# EPICS substitutions: siteApps/alarmPerfTest/alarmTestApp/Db/alarm.substitutions
###############################
file "$(DB_TOP)/alarm.template" { pattern
{S,				VAL}
{Alarm0,			92.30}
{Alarm1,			95.71}
{Alarm2,			98.12}
{Alarm3,			91.53}
{Alarm4,			94.94}
{Alarm5,			97.35}
{Alarm6,			90.76}
{Alarm7,			93.17}
{Alarm8,			96.58}
{Alarm9,			99.99}
{Alarm10,			92.30}
{Alarm11,			95.71}
{Alarm12,			98.12}
{Alarm13,			91.53}
{Alarm14,			94.94}
{Alarm15,			97.35}
{Alarm16,			90.76}
{Alarm17,			93.17}
{Alarm18,			96.58}
{Alarm19,			99.99}
{Alarm20,			92.30}
{Alarm21,			95.71}
{Alarm22,			98.12}
{Alarm23,			91.53}
{Alarm24,			94.94}
{Alarm25,			97.35}
{Alarm26,			90.76}
{Alarm27,			93.17}
{Alarm28,			96.58}
{Alarm29,			99.99}
{Alarm30,			92.30}
{Alarm31,			95.71}
{Alarm32,			98.02}
{Alarm33,			91.03}
{Alarm34,			94.04}
{Alarm35,			97.15}
{Alarm36,			90.16}
{Alarm37,			93.27}
{Alarm38,			96.28}
{Alarm39,			99.29}
{Alarm40,			92.20}
{Alarm41,			95.21}
{Alarm42,			98.32}
{Alarm43,			91.33}
{Alarm44,			99.34}
{Alarm45,			99.45}
{Alarm46,			90.46}
{Alarm47,			93.57}
{Alarm48,			96.58}
{Alarm49,			99.59}
{Alarm50,			92.50}
{Alarm51,			95.51}
{Alarm52,			98.62}
{Alarm53,			91.63}
{Alarm54,			94.64}
{Alarm55,			97.75}
{Alarm56,			90.76}
{Alarm57,			93.87}
{Alarm58,			96.88}
{Alarm59,			99.89}
{Alarm60,			92.80}
{Alarm61,			95.81}
{Alarm62,			98.92}
{Alarm63,			91.93}
{Alarm64,			94.94}
{Alarm65,			97.05}
{Alarm66,			90.06}
{Alarm67,			93.17}
{Alarm68,			96.18}
{Alarm69,			99.19}
{Alarm70,			92.10}
{Alarm71,			95.11}
{Alarm72,			98.22}
{Alarm73,			91.23}
{Alarm74,			94.24}
{Alarm75,			97.35}
{Alarm76,			90.36}
{Alarm77,			93.47}
{Alarm78,			96.48}
{Alarm79,			99.49}
{Alarm80,			92.40}
{Alarm81,			95.41}
{Alarm82,			98.52}
{Alarm83,			91.53}
{Alarm84,			94.54}
{Alarm85,			97.65}
{Alarm86,			90.66}
{Alarm87,			93.77}
{Alarm88,			96.78}
{Alarm89,			99.79}
{Alarm90,			92.70}
{Alarm91,			95.71}
{Alarm92,			98.82}
{Alarm93,			91.83}
{Alarm94,			94.84}
{Alarm95,			97.95}
{Alarm96,			90.96}
{Alarm97,			93.07}
{Alarm98,			96.08}
{Alarm99,			99.09}
{Alarm100,			92.00}
{Alarm101,			95.01}
{Alarm102,			98.12}
{Alarm103,			91.13}
{Alarm104,			94.14}
{Alarm105,			97.25}
{Alarm106,			90.26}
{Alarm107,			93.37}
{Alarm108,			96.38}
{Alarm109,			99.39}
{Alarm110,			92.30}
{Alarm111,			95.31}
{Alarm112,			98.42}
{Alarm113,			91.43}
{Alarm114,			94.44}
{Alarm115,			97.55}
{Alarm116,			90.56}
{Alarm117,			93.67}
{Alarm118,			96.68}
{Alarm119,			99.69}
{Alarm120,			92.60}
{Alarm121,			95.61}
{Alarm122,			98.72}
{Alarm123,			91.73}
{Alarm124,			94.74}
{Alarm125,			97.85}
{Alarm126,			90.86}
{Alarm127,			93.97}
{Alarm128,			96.98}
{Alarm129,			99.99}
{Alarm130,			92.90}
{Alarm131,			95.91}
{Alarm132,			98.02}
{Alarm133,			91.03}
{Alarm134,			94.04}
{Alarm135,			97.15}
{Alarm136,			90.16}
{Alarm137,			93.27}
{Alarm138,			96.28}
{Alarm139,			99.29}
{Alarm140,			92.20}
{Alarm141,			95.21}
{Alarm142,			98.32}
{Alarm143,			91.33}
{Alarm144,			94.34}
{Alarm145,			97.45}
{Alarm146,			90.46}
{Alarm147,			93.57}
{Alarm148,			96.58}
{Alarm149,			99.59}
{Alarm150,			92.50}
{Alarm151,			95.51}
{Alarm152,			98.62}
{Alarm153,			91.63}
{Alarm154,			94.64}
{Alarm155,			97.75}
{Alarm156,			90.76}
{Alarm157,			93.87}
{Alarm158,			96.88}
{Alarm159,			99.89}
{Alarm160,			92.80}
{Alarm161,			95.81}
{Alarm162,			98.92}
{Alarm163,			91.93}
{Alarm164,			94.94}
{Alarm165,			97.05}
{Alarm166,			90.06}
{Alarm167,			93.17}
{Alarm168,			96.18}
{Alarm169,			99.19}
{Alarm170,			92.10}
{Alarm171,			95.11}
{Alarm172,			98.22}
{Alarm173,			91.23}
{Alarm174,			94.24}
{Alarm175,			97.35}
{Alarm176,			90.36}
{Alarm177,			93.47}
{Alarm178,			96.48}
{Alarm179,			99.49}
{Alarm180,			92.40}
{Alarm181,			95.41}
{Alarm182,			98.52}
{Alarm183,			91.53}
{Alarm184,			94.54}
{Alarm185,			97.65}
{Alarm186,			90.66}
{Alarm187,			93.77}
{Alarm188,			96.78}
{Alarm189,			99.79}
{Alarm190,			92.70}
{Alarm191,			95.71}
{Alarm192,			98.82}
{Alarm193,			91.83}
{Alarm194,			94.84}
{Alarm195,			97.95}
{Alarm196,			90.96}
{Alarm197,			93.07}
{Alarm198,			96.08}
{Alarm199,			99.09}
{Alarm200,			92.00}
{Alarm201,			95.01}
{Alarm202,			98.12}
{Alarm203,			91.13}
{Alarm204,			94.14}
{Alarm205,			97.25}
{Alarm206,			90.26}
{Alarm207,			93.37}
{Alarm208,			96.38}
{Alarm209,			99.39}
{Alarm210,			92.30}
{Alarm211,			95.31}
{Alarm212,			98.42}
{Alarm213,			91.43}
{Alarm214,			94.44}
{Alarm215,			97.55}
{Alarm216,			90.56}
{Alarm217,			93.67}
{Alarm218,			96.68}
{Alarm219,			99.69}
{Alarm220,			92.60}
{Alarm221,			95.61}
{Alarm222,			98.72}
{Alarm223,			91.73}
{Alarm224,			94.74}
{Alarm225,			97.85}
{Alarm226,			90.86}
{Alarm227,			93.97}
{Alarm228,			96.98}
{Alarm229,			99.99}
{Alarm230,			92.90}
{Alarm231,			95.91}
{Alarm232,			98.02}
{Alarm233,			91.03}
{Alarm234,			94.04}
{Alarm235,			97.15}
{Alarm236,			90.16}
{Alarm237,			93.27}
{Alarm238,			96.28}
{Alarm239,			99.29}
{Alarm240,			92.20}
{Alarm241,			95.21}
{Alarm242,			98.32}
{Alarm243,			91.33}
{Alarm244,			94.34}
{Alarm245,			97.45}
{Alarm246,			90.46}
{Alarm247,			93.57}
{Alarm248,			96.58}
{Alarm249,			99.59}
{Alarm250,			92.50}
{Alarm251,			95.51}
{Alarm252,			98.62}
{Alarm253,			91.63}
{Alarm254,			94.64}
{Alarm255,			97.75}
{Alarm256,			90.76}
{Alarm257,			93.87}
{Alarm258,			96.88}
{Alarm259,			99.89}
{Alarm260,			92.80}
{Alarm261,			95.81}
{Alarm262,			98.92}
{Alarm263,			91.93}
{Alarm264,			94.94}
{Alarm265,			97.05}
{Alarm266,			90.06}
{Alarm267,			93.17}
{Alarm268,			96.18}
{Alarm269,			99.19}
{Alarm270,			92.10}
{Alarm271,			95.11}
{Alarm272,			98.22}
{Alarm273,			91.23}
{Alarm274,			94.24}
{Alarm275,			97.35}
{Alarm276,			90.36}
{Alarm277,			93.47}
{Alarm278,			96.48}
{Alarm279,			99.49}
{Alarm280,			92.40}
{Alarm281,			95.41}
{Alarm282,			98.52}
{Alarm283,			91.53}
{Alarm284,			94.54}
{Alarm285,			97.65}
{Alarm286,			90.66}
{Alarm287,			93.77}
{Alarm288,			96.78}
{Alarm289,			99.79}
{Alarm290,			92.70}
{Alarm291,			95.71}
{Alarm292,			98.82}
{Alarm293,			91.83}
{Alarm294,			94.84}
{Alarm295,			97.95}
{Alarm296,			90.96}
{Alarm297,			93.07}
{Alarm298,			96.08}
{Alarm299,			99.09}
{Alarm300,			92.00}
{Alarm301,			95.01}
{Alarm302,			98.12}
{Alarm303,			91.13}
{Alarm304,			94.14}
{Alarm305,			97.25}
{Alarm306,			90.26}
{Alarm307,			93.37}
{Alarm308,			96.38}
{Alarm309,			99.39}
{Alarm310,			92.30}
{Alarm311,			95.31}
{Alarm312,			98.42}
{Alarm313,			91.43}
{Alarm314,			94.44}
{Alarm315,			97.55}
{Alarm316,			90.56}
{Alarm317,			93.67}
{Alarm318,			96.68}
{Alarm319,			99.69}
{Alarm320,			92.60}
{Alarm321,			95.61}
{Alarm322,			98.72}
{Alarm323,			91.73}
{Alarm324,			94.74}
{Alarm325,			97.85}
{Alarm326,			90.86}
{Alarm327,			93.97}
{Alarm328,			96.98}
{Alarm329,			99.99}
{Alarm330,			92.90}
{Alarm331,			95.91}
{Alarm332,			98.12}
{Alarm333,			91.53}
{Alarm334,			94.94}
{Alarm335,			97.35}
{Alarm336,			90.76}
{Alarm337,			93.17}
{Alarm338,			96.58}
{Alarm339,			99.99}
{Alarm340,			92.30}
{Alarm341,			95.71}
{Alarm342,			98.12}
{Alarm343,			91.53}
{Alarm344,			94.94}
{Alarm345,			97.35}
{Alarm346,			90.76}
{Alarm347,			93.17}
{Alarm348,			96.58}
{Alarm349,			99.99}
{Alarm350,			92.30}
{Alarm351,			95.71}
{Alarm352,			98.12}
{Alarm353,			91.53}
{Alarm354,			94.94}
{Alarm355,			97.35}
{Alarm356,			90.76}
{Alarm357,			93.17}
{Alarm358,			96.58}
{Alarm359,			99.99}
{Alarm360,			92.30}
{Alarm361,			95.71}
{Alarm362,			98.12}
{Alarm363,			91.53}
{Alarm364,			94.94}
{Alarm365,			97.35}
{Alarm366,			90.76}
{Alarm367,			93.17}
{Alarm368,			96.58}
{Alarm369,			99.99}
{Alarm370,			92.30}
{Alarm371,			95.71}
{Alarm372,			98.12}
{Alarm373,			91.53}
{Alarm374,			94.94}
{Alarm375,			97.35}
{Alarm376,			90.76}
{Alarm377,			93.17}
{Alarm378,			96.58}
{Alarm379,			99.99}
{Alarm380,			92.30}
{Alarm381,			95.71}
{Alarm382,			98.12}
{Alarm383,			91.53}
{Alarm384,			94.94}
{Alarm385,			97.35}
{Alarm386,			90.76}
{Alarm387,			93.17}
{Alarm388,			96.58}
{Alarm389,			99.99}
{Alarm390,			92.30}
{Alarm391,			95.71}
{Alarm392,			98.12}
{Alarm393,			91.53}
{Alarm394,			94.94}
{Alarm395,			97.35}
{Alarm396,			90.76}
{Alarm397,			93.17}
{Alarm398,			96.58}
{Alarm399,			99.99}
{Alarm400,			92.30}
{Alarm401,			95.71}
{Alarm402,			98.12}
{Alarm403,			91.53}
{Alarm404,			94.94}
{Alarm405,			97.35}
{Alarm406,			90.76}
{Alarm407,			93.17}
{Alarm408,			96.58}
{Alarm409,			99.99}
{Alarm410,			92.30}
{Alarm411,			95.71}
{Alarm412,			98.12}
{Alarm413,			91.53}
{Alarm414,			94.94}
{Alarm415,			97.35}
{Alarm416,			90.76}
{Alarm417,			93.17}
{Alarm418,			96.58}
{Alarm419,			99.99}
{Alarm420,			92.30}
{Alarm421,			95.71}
{Alarm422,			98.12}
{Alarm423,			91.53}
{Alarm424,			94.94}
{Alarm425,			97.35}
{Alarm426,			90.76}
{Alarm427,			93.17}
{Alarm428,			96.58}
{Alarm429,			99.99}
{Alarm430,			92.30}
{Alarm431,			95.71}
{Alarm432,			98.12}
{Alarm433,			91.53}
{Alarm434,			94.94}
{Alarm435,			97.35}
{Alarm436,			90.76}
{Alarm437,			93.17}
{Alarm438,			96.58}
{Alarm439,			99.99}
{Alarm440,			92.30}
{Alarm441,			95.71}
{Alarm442,			98.12}
{Alarm443,			91.53}
{Alarm444,			94.94}
{Alarm445,			97.35}
{Alarm446,			90.76}
{Alarm447,			93.17}
{Alarm448,			96.58}
{Alarm449,			99.99}
{Alarm450,			92.30}
{Alarm451,			95.71}
{Alarm452,			98.12}
{Alarm453,			91.53}
{Alarm454,			94.94}
{Alarm455,			97.35}
{Alarm456,			90.76}
{Alarm457,			93.17}
{Alarm458,			96.58}
{Alarm459,			99.99}
{Alarm460,			92.30}
{Alarm461,			95.71}
{Alarm462,			98.12}
{Alarm463,			91.53}
{Alarm464,			94.94}
{Alarm465,			97.35}
{Alarm466,			90.76}
{Alarm467,			93.17}
{Alarm468,			96.58}
{Alarm469,			99.99}
{Alarm470,			92.30}
{Alarm471,			95.71}
{Alarm472,			98.12}
{Alarm473,			91.53}
{Alarm474,			94.94}
{Alarm475,			97.35}
{Alarm476,			90.76}
{Alarm477,			93.17}
{Alarm478,			96.58}
{Alarm479,			99.99}
{Alarm480,			92.30}
{Alarm481,			95.71}
{Alarm482,			98.12}
{Alarm483,			91.53}
{Alarm484,			94.94}
{Alarm485,			97.35}
{Alarm486,			90.76}
{Alarm487,			93.17}
{Alarm488,			96.58}
{Alarm489,			99.99}
{Alarm490,			92.30}
{Alarm491,			95.71}
{Alarm492,			98.12}
{Alarm493,			91.53}
{Alarm494,			94.94}
{Alarm495,			97.35}
{Alarm496,			90.76}
{Alarm497,			93.17}
{Alarm498,			96.58}
{Alarm499,			99.99}
{Alarm500,			92.30}
{Alarm501,			95.71}
{Alarm502,			98.12}
{Alarm503,			91.53}
{Alarm504,			94.94}
{Alarm505,			97.35}
{Alarm506,			90.76}
{Alarm507,			93.17}
{Alarm508,			96.58}
{Alarm509,			99.99}
{Alarm510,			92.30}
{Alarm511,			95.71}
{Alarm512,			98.12}
{Alarm513,			91.53}
{Alarm514,			94.94}
{Alarm515,			97.35}
{Alarm516,			90.76}
{Alarm517,			93.17}
{Alarm518,			96.58}
{Alarm519,			99.99}
{Alarm520,			92.30}
{Alarm521,			95.71}
{Alarm522,			98.12}
{Alarm523,			91.53}
{Alarm524,			94.94}
{Alarm525,			97.35}
{Alarm526,			90.76}
{Alarm527,			93.17}
{Alarm528,			96.58}
{Alarm529,			99.99}
{Alarm530,			92.30}
{Alarm531,			95.71}
{Alarm532,			98.12}
{Alarm533,			91.53}
{Alarm534,			94.94}
{Alarm535,			97.35}
{Alarm536,			90.76}
{Alarm537,			93.17}
{Alarm538,			96.58}
{Alarm539,			99.99}
{Alarm540,			92.30}
{Alarm541,			95.71}
{Alarm542,			98.12}
{Alarm543,			91.53}
{Alarm544,			94.94}
{Alarm545,			97.35}
{Alarm546,			90.76}
{Alarm547,			93.17}
{Alarm548,			96.58}
{Alarm549,			99.99}
{Alarm550,			92.30}
{Alarm551,			95.71}
{Alarm552,			98.12}
{Alarm553,			91.53}
{Alarm554,			94.94}
{Alarm555,			97.35}
{Alarm556,			90.76}
{Alarm557,			93.17}
{Alarm558,			96.58}
{Alarm559,			99.99}
{Alarm560,			92.30}
{Alarm561,			95.71}
{Alarm562,			98.12}
{Alarm563,			91.53}
{Alarm564,			94.94}
{Alarm565,			97.35}
{Alarm566,			90.76}
{Alarm567,			93.17}
{Alarm568,			96.58}
{Alarm569,			99.99}
{Alarm570,			92.30}
{Alarm571,			95.71}
{Alarm572,			98.12}
{Alarm573,			91.53}
{Alarm574,			94.94}
{Alarm575,			97.35}
{Alarm576,			90.76}
{Alarm577,			93.17}
{Alarm578,			96.58}
{Alarm579,			99.99}
{Alarm580,			92.30}
{Alarm581,			95.71}
{Alarm582,			98.12}
{Alarm583,			91.53}
{Alarm584,			94.94}
{Alarm585,			97.35}
{Alarm586,			90.76}
{Alarm587,			93.17}
{Alarm588,			96.58}
{Alarm589,			99.99}
{Alarm590,			92.30}
{Alarm591,			95.71}
{Alarm592,			98.12}
{Alarm593,			91.53}
{Alarm594,			94.94}
{Alarm595,			97.35}
{Alarm596,			90.76}
{Alarm597,			93.17}
{Alarm598,			96.58}
{Alarm599,			99.99}
{Alarm600,			92.30}
{Alarm601,			95.71}
{Alarm602,			98.12}
{Alarm603,			91.53}
{Alarm604,			94.94}
{Alarm605,			97.35}
{Alarm606,			90.76}
{Alarm607,			93.17}
{Alarm608,			96.58}
{Alarm609,			99.99}
{Alarm610,			92.30}
{Alarm611,			95.71}
{Alarm612,			98.12}
{Alarm613,			91.53}
{Alarm614,			94.94}
{Alarm615,			97.35}
{Alarm616,			90.76}
{Alarm617,			93.17}
{Alarm618,			96.58}
{Alarm619,			99.99}
{Alarm620,			92.30}
{Alarm621,			95.71}
{Alarm622,			98.12}
{Alarm623,			91.53}
{Alarm624,			94.94}
{Alarm625,			97.35}
{Alarm626,			90.76}
{Alarm627,			93.17}
{Alarm628,			96.58}
{Alarm629,			99.99}
{Alarm630,			92.30}
{Alarm631,			95.71}
{Alarm632,			98.12}
{Alarm633,			91.53}
{Alarm634,			94.94}
{Alarm635,			97.35}
{Alarm636,			90.76}
{Alarm637,			93.17}
{Alarm638,			96.58}
{Alarm639,			99.99}
{Alarm640,			92.30}
{Alarm641,			95.71}
{Alarm642,			98.12}
{Alarm643,			91.53}
{Alarm644,			94.94}
{Alarm645,			97.35}
{Alarm646,			90.76}
{Alarm647,			93.17}
{Alarm648,			96.58}
{Alarm649,			99.99}
{Alarm650,			92.30}
{Alarm651,			95.71}
{Alarm652,			98.12}
{Alarm653,			91.53}
{Alarm654,			94.94}
{Alarm655,			97.35}
{Alarm656,			90.76}
{Alarm657,			93.17}
{Alarm658,			96.58}
{Alarm659,			99.99}
{Alarm660,			92.30}
{Alarm661,			95.71}
{Alarm662,			98.12}
{Alarm663,			91.53}
{Alarm664,			94.94}
{Alarm665,			97.35}
{Alarm666,			90.76}
{Alarm667,			93.17}
{Alarm668,			96.58}
{Alarm669,			99.99}
{Alarm670,			92.30}
{Alarm671,			95.71}
{Alarm672,			98.12}
{Alarm673,			91.53}
{Alarm674,			94.94}
{Alarm675,			97.35}
{Alarm676,			90.76}
{Alarm677,			93.17}
{Alarm678,			96.58}
{Alarm679,			99.99}
{Alarm680,			92.30}
{Alarm681,			95.71}
{Alarm682,			98.12}
{Alarm683,			91.53}
{Alarm684,			94.94}
{Alarm685,			97.35}
{Alarm686,			90.76}
{Alarm687,			93.17}
{Alarm688,			96.58}
{Alarm689,			99.99}
{Alarm690,			92.30}
{Alarm691,			95.71}
{Alarm692,			98.12}
{Alarm693,			91.53}
{Alarm694,			94.94}
{Alarm695,			97.35}
{Alarm696,			90.76}
{Alarm697,			93.17}
{Alarm698,			96.58}
{Alarm699,			99.99}
{Alarm700,			92.30}
{Alarm701,			95.71}
{Alarm702,			98.12}
{Alarm703,			91.53}
{Alarm704,			94.94}
{Alarm705,			97.35}
{Alarm706,			90.76}
{Alarm707,			93.17}
{Alarm708,			96.58}
{Alarm709,			99.99}
{Alarm710,			92.30}
{Alarm711,			95.71}
{Alarm712,			98.12}
{Alarm713,			91.53}
{Alarm714,			94.94}
{Alarm715,			97.35}
{Alarm716,			90.76}
{Alarm717,			93.17}
{Alarm718,			96.58}
{Alarm719,			99.99}
{Alarm720,			92.30}
{Alarm721,			95.71}
{Alarm722,			98.12}
{Alarm723,			91.53}
{Alarm724,			94.94}
{Alarm725,			97.35}
{Alarm726,			90.76}
{Alarm727,			93.17}
{Alarm728,			96.58}
{Alarm729,			99.99}
{Alarm730,			92.30}
{Alarm731,			95.71}
{Alarm732,			98.12}
{Alarm733,			91.53}
{Alarm734,			94.94}
{Alarm735,			97.35}
{Alarm736,			90.76}
{Alarm737,			93.17}
{Alarm738,			96.58}
{Alarm739,			99.99}
{Alarm740,			92.30}
{Alarm741,			95.71}
{Alarm742,			98.12}
{Alarm743,			91.53}
{Alarm744,			94.94}
{Alarm745,			97.35}
{Alarm746,			90.76}
{Alarm747,			93.17}
{Alarm748,			96.58}
{Alarm749,			99.99}
{Alarm750,			92.30}
{Alarm751,			95.71}
{Alarm752,			98.12}
{Alarm753,			91.53}
{Alarm754,			94.94}
{Alarm755,			97.35}
{Alarm756,			90.76}
{Alarm757,			93.17}
{Alarm758,			96.58}
{Alarm759,			99.99}
{Alarm760,			92.30}
{Alarm761,			95.71}
{Alarm762,			98.12}
{Alarm763,			91.53}
{Alarm764,			94.94}
{Alarm765,			97.35}
{Alarm766,			90.76}
{Alarm767,			93.17}
{Alarm768,			96.58}
{Alarm769,			99.99}
{Alarm770,			92.30}
{Alarm771,			95.71}
{Alarm772,			98.12}
{Alarm773,			91.53}
{Alarm774,			94.94}
{Alarm775,			97.35}
{Alarm776,			90.76}
{Alarm777,			93.17}
{Alarm778,			96.58}
{Alarm779,			99.99}
{Alarm780,			92.30}
{Alarm781,			95.71}
{Alarm782,			98.12}
{Alarm783,			91.53}
{Alarm784,			94.94}
{Alarm785,			97.35}
{Alarm786,			90.76}
{Alarm787,			93.17}
{Alarm788,			96.58}
{Alarm789,			99.99}
{Alarm790,			92.30}
{Alarm791,			95.71}
{Alarm792,			98.12}
{Alarm793,			91.53}
{Alarm794,			94.94}
{Alarm795,			97.35}
{Alarm796,			90.76}
{Alarm797,			93.17}
{Alarm798,			96.58}
{Alarm799,			99.99}
{Alarm800,			92.30}
{Alarm801,			95.71}
{Alarm802,			98.12}
{Alarm803,			91.53}
{Alarm804,			94.94}
{Alarm805,			97.35}
{Alarm806,			90.76}
{Alarm807,			93.17}
{Alarm808,			96.58}
{Alarm809,			99.99}
{Alarm810,			92.30}
{Alarm811,			95.71}
{Alarm812,			98.12}
{Alarm813,			91.53}
{Alarm814,			94.94}
{Alarm815,			97.35}
{Alarm816,			90.76}
{Alarm817,			93.17}
{Alarm818,			96.58}
{Alarm819,			99.99}
{Alarm820,			92.30}
{Alarm821,			95.71}
{Alarm822,			98.12}
{Alarm823,			91.53}
{Alarm824,			94.94}
{Alarm825,			97.35}
{Alarm826,			90.76}
{Alarm827,			93.17}
{Alarm828,			96.58}
{Alarm829,			99.99}
{Alarm830,			92.30}
{Alarm831,			95.71}
{Alarm832,			98.12}
{Alarm833,			91.53}
{Alarm834,			94.94}
{Alarm835,			97.35}
{Alarm836,			90.76}
{Alarm837,			93.17}
{Alarm838,			96.58}
{Alarm839,			99.99}
{Alarm840,			92.30}
{Alarm841,			95.71}
{Alarm842,			98.12}
{Alarm843,			91.53}
{Alarm844,			94.94}
{Alarm845,			97.35}
{Alarm846,			90.76}
{Alarm847,			93.17}
{Alarm848,			96.58}
{Alarm849,			99.99}
{Alarm850,			92.30}
{Alarm851,			95.71}
{Alarm852,			98.12}
{Alarm853,			91.53}
{Alarm854,			94.94}
{Alarm855,			97.35}
{Alarm856,			90.76}
{Alarm857,			93.17}
{Alarm858,			96.58}
{Alarm859,			99.99}
{Alarm860,			92.30}
{Alarm861,			95.71}
{Alarm862,			98.12}
{Alarm863,			91.53}
{Alarm864,			94.94}
{Alarm865,			97.35}
{Alarm866,			90.76}
{Alarm867,			93.17}
{Alarm868,			96.58}
{Alarm869,			99.99}
{Alarm870,			92.30}
{Alarm871,			95.71}
{Alarm872,			98.12}
{Alarm873,			91.53}
{Alarm874,			94.94}
{Alarm875,			97.35}
{Alarm876,			90.76}
{Alarm877,			93.17}
{Alarm878,			96.58}
{Alarm879,			99.99}
{Alarm880,			92.30}
{Alarm881,			95.71}
{Alarm882,			98.12}
{Alarm883,			91.53}
{Alarm884,			94.94}
{Alarm885,			97.35}
{Alarm886,			90.76}
{Alarm887,			93.17}
{Alarm888,			96.58}
{Alarm889,			99.99}
{Alarm890,			92.30}
{Alarm891,			95.71}
{Alarm892,			98.12}
{Alarm893,			91.53}
{Alarm894,			94.94}
{Alarm895,			97.35}
{Alarm896,			90.76}
{Alarm897,			93.17}
{Alarm898,			96.58}
{Alarm899,			99.99}
{Alarm900,			92.30}
{Alarm901,			95.71}
{Alarm902,			98.12}
{Alarm903,			91.53}
{Alarm904,			94.94}
{Alarm905,			97.35}
{Alarm906,			90.76}
{Alarm907,			93.17}
{Alarm908,			96.58}
{Alarm909,			99.99}
{Alarm910,			92.30}
{Alarm911,			95.71}
{Alarm912,			98.12}
{Alarm913,			91.53}
{Alarm914,			94.94}
{Alarm915,			97.35}
{Alarm916,			90.76}
{Alarm917,			93.17}
{Alarm918,			96.58}
{Alarm919,			99.99}
{Alarm920,			92.30}
{Alarm921,			95.71}
{Alarm922,			98.12}
{Alarm923,			91.53}
{Alarm924,			94.94}
{Alarm925,			97.35}
{Alarm926,			90.76}
{Alarm927,			93.17}
{Alarm928,			96.58}
{Alarm929,			99.99}
{Alarm930,			92.30}
{Alarm931,			95.71}
{Alarm932,			98.12}
{Alarm933,			91.53}
{Alarm934,			94.94}
{Alarm935,			97.35}
{Alarm936,			90.76}
{Alarm937,			93.17}
{Alarm938,			96.58}
{Alarm939,			99.99}
{Alarm940,			92.30}
{Alarm941,			95.71}
{Alarm942,			98.12}
{Alarm943,			91.53}
{Alarm944,			94.94}
{Alarm945,			97.35}
{Alarm946,			90.76}
{Alarm947,			93.17}
{Alarm948,			96.58}
{Alarm949,			99.99}
{Alarm950,			92.30}
{Alarm951,			95.71}
{Alarm952,			98.12}
{Alarm953,			91.53}
{Alarm954,			94.94}
{Alarm955,			97.35}
{Alarm956,			90.76}
{Alarm957,			93.17}
{Alarm958,			96.58}
{Alarm959,			99.99}
{Alarm960,			92.30}
{Alarm961,			95.71}
{Alarm962,			98.12}
{Alarm963,			91.53}
{Alarm964,			94.94}
{Alarm965,			97.35}
{Alarm966,			90.76}
{Alarm967,			93.17}
{Alarm968,			96.58}
{Alarm969,			99.99}
{Alarm970,			92.30}
{Alarm971,			95.71}
{Alarm972,			98.12}
{Alarm973,			91.53}
{Alarm974,			94.94}
{Alarm975,			97.35}
{Alarm976,			90.76}
{Alarm977,			93.17}
{Alarm978,			96.58}
{Alarm979,			99.99}
{Alarm980,			92.30}
{Alarm981,			95.71}
{Alarm982,			98.12}
{Alarm983,			91.53}
{Alarm984,			94.94}
{Alarm985,			97.35}
{Alarm986,			90.76}
{Alarm987,			93.17}
{Alarm988,			96.58}
{Alarm989,			99.99}
{Alarm990,			92.30}
{Alarm991,			95.71}
{Alarm992,			98.12}
{Alarm993,			91.53}
{Alarm994,			94.94}
{Alarm995,			97.35}
{Alarm996,			90.76}
{Alarm997,			93.17}
{Alarm998,			96.58}
{Alarm999,			99.99}
}
